(* IEC 61131-3 sources: CodesysTest/alpha/export/ObjectHandling/IMachineLogger.itf, 1 file *)

(* ---- AddLogItem.m.st ---- *)
(*#-#-#-#-#-#-#-#-#-#---Declaration---#-#-#-#-#-#-#-#-#-#-#-#-#*)

METHOD AddLogItem
VAR_INPUT
	message : STRING;
END_VAR
